FUNCTION_BLOCK FB_DXL_XL
VAR_INPUT 
	id : INT;
END_VAR
VAR  
	//communication en cours
	com_ongoing	: BOOL;
END_VAR
VAR CONSTANT
	//type du moteur
	XL430:USINT:=2;
	AX12A:USINT:=1;
	
	motor_type : USINT:=XL430;
END_VAR

//author: Alec Horth
//mail  : horth.alec@gmail.com

METHOD PRIVATE _end_communication : BOOL
VAR_IN_OUT
	run:BOOL; // arrête la variable qui maintient la fonction en vie 
	started:BOOL; // arrête la variable qui indique que la fonction possède un token
END_VAR
VAR_INST
	pulse : F_TRIG;
	once : bool;
END_VAR
// front descendant activé par le script python et désactivé par la fonction _send()
// confirme que la commande à bien été envoyée
pulse(CLK:=G_DXL.bDone AND started, Q=>);

IF pulse.Q THEN 
	//permet de lancer cette fonction une seule fois, sinon elle relance un cycle de façon involontaire 
	once := TRUE;
END_IF

IF once THEN
	// libère le token
	G_DXL.bToken := G_DXL.iOPEN_TOKEN;
	com_ongoing := FALSE;
	run := FALSE;
	_end_communication := TRUE;
	started := FALSE;
	once := FALSE;
ELSE
	_end_communication := FALSE;
END_IF
END_METHOD

METHOD PRIVATE _send : BOOL
VAR_INPUT
END_VAR
VAR_INST
	once :BOOL; // assure que la commande n'est envoyé qu'une fois
END_VAR
IF G_DXL.bDone THEN 	//confirmation d'acquisition de la commande du script python
	G_DXL.bRun := FALSE; //indique au script python que le message est passé
ELSIF NOT G_DXL.bDone AND NOT once THEN // si la commande n'a pas encore été envoyé, lance la commande
	once := TRUE;
	G_DXL.bRun := TRUE;
END_IF

IF NOT com_ongoing THEN // permet de relancer des commandes lorsque le token est rendu
	once := FALSE;
END_IF
END_METHOD

METHOD PRIVATE _start_communication : BOOL
VAR_IN_OUT
	started:BOOL; //maintient la fonction active tant que le token n'est pas rendu
END_VAR
IF ((G_DXL.bToken = G_DXL.iOPEN_TOKEN OR G_DXL.bToken = id) AND NOT com_ongoing AND NOT G_DXL.bDone) OR started THEN // vérifie que tous les token soient libres
	// attribution du token
	started := TRUE; 
	G_DXL.bToken := id;
	// configure les commandes à envoyer avec le bon ID et le bon type du moteur
	G_DXL.iID := id;
	G_DXL.usiMotor_type := motor_type;
	com_ongoing := TRUE; 
	_start_communication := TRUE;	
ELSE 
	_start_communication := FALSE;
END_IF
END_METHOD

METHOD private BASE_EXEMPLE_FUTUR_MODIF_SEND : BOOL
VAR_INPUT
	EN			:BOOL; // un front montant change le taux d'accélération du moteur
	
	//--------------TO DO---------------
	parametre1	:usint;
	parametre2	:INT;
	//----------------------------------

END_VAR
VAR_OUTPUT
	done		:BOOL; //la commande est envoyée, passe à False si EN passe aussi à False
END_VAR
VAR_INST 
	bRun 		:BOOL;
	rtrigPulse 	:R_TRIG;
	bDone_pulse :BOOL;
	bStarted 	:BOOL;
END_VAR
// IL EST POSSIBLE DE MODIFIER LES SECTION "TO DO", LE RESTE NE DOIT PAS ÊTRE MODIFIE

//Activation de la fonction
rtrigPulse(CLK:=EN, Q=>);

IF rtrigPulse.Q THEN
	//Si une autre fonction est déjà en cours de traitement (token déjà pris) cette fonction ne peut pas être effectuée
	//La variable run garde l'ordre d'activation en mémoire et lance la fonction dès que le token est libéré
	bRun := TRUE;
END_IF

IF bRun THEN
	IF _start_communication(started:=bStarted) THEN 	//vérifie si les tokens sont libérés 
		
		//--------------TO DO---------------
		G_DXL.usiFonction := G_DXL.usiGOAL_ACCELERATION; 	// choix de la commande à envoyer		
		G_DXL.usiAcceleration 	:= parametre1;				//paramètre 1
		G_DXL.iSpeed    		:= parametre2;				//paramètre 2 
		//----------------------------------
		
		
		bDone_pulse := _end_communication(run:=bRun, started:=bStarted) AND EN;	//libère le token une fois que la commande est lancée
		_send();																//Envoi de la commande au moteur
	END_IF
END_IF;

IF bDone_pulse AND EN THEN														//Affiche le status d'excution de la fonction
	done := EN;																	//tant que EN est à True
ELSIF bDone_pulse AND NOT EN THEN
	bDone_pulse := FALSE;
END_IF
END_METHOD

METHOD get_load 
VAR_INPUT
	EN:BOOL; 	// ouvre un canal de transmission avec le moteur 
END_VAR
VAR_OUTPUT
	load:INT; 	// le moteur renvoie le torque qu'il emet à travers le canal (voir dans la méthode pour + d'infos)
				//(AX12A) 0-1023 torque est dans le sens inverse des aiguilles d'une montre, entre 1024 et 2047 le torque est dans le sens des aiguilles d'une montre
				//(XL430) +- 1000 pour mille du torque maximum si la valeur est positive => le torque est dans le sens inverse des aiguilles d'une montre
	done:bool;
END_VAR
VAR_inst 
	run :BOOL;
	pulse : R_TRIG;
	started: BOOL;
END_VAR
//ouvre le canal de transmission
pulse(CLK:=EN, Q=>);

IF pulse.Q THEN
	//Si une autre fonction est déjà en cours de traitement (token déjà pris) le canal ne peut pas être ouvert
	//La variable run garde l'ordre d'activation en mémoire et ouvre le canal dès que le token est libéré
	run := TRUE;
END_IF

IF run THEN 
	IF _start_communication(started := started) THEN 	// Vérifie si le token est libre
		G_DXL.usiFonction := G_DXL.usiGET_PRESENT_LOAD;	// configure le canal à ouvrir
		G_DXL.bRun := TRUE;								// envoie la commande au script python
		load := G_DXL.iDxl_load;						// si le canal est ouvert, renvoie la valeur actuelle du torque émit pas le moteur
	END_IF
	IF NOT EN THEN
		G_DXL.bRun 	:= FALSE;						    //ferme le canal
		G_DXL.iDxl_load := -9000;						//remet une valeur par défault
		_end_communication(run:=run,started := started);//libère le token
	END_IF;
ELSE
	load := -9000;										//valeur par défaut
END_IF
END_METHOD

METHOD get_movement 
VAR_INPUT
	EN:BOOL; 	// ouvre un canal de transmission avec le moteur 
END_VAR
VAR_OUTPUT
	mouvement:BOOL; // le moteur renvoie si il est en mouvement(TRUE) ou non (FALSE)
END_VAR
VAR_INST 
	run :BOOL;
	pulse : R_TRIG;
	started: BOOL;
END_VAR
//ouvre le canal de transmission
pulse(CLK:=EN, Q=>);

IF pulse.Q THEN
	//Si une autre fonction est déjà en cours de traitement (token déjà pris) le canal ne peut pas être ouvert
	//La variable run garde l'ordre d'activation en mémoire et ouvre le canal dès que le token est libéré
	run := TRUE;
END_IF

IF run THEN 
	IF _start_communication(started := started) THEN 	// Vérifie si le token est libre
		G_DXL.usiFonction := G_DXL.usiGET_PRESENT_MOVEMENT;	// configure le canal à ouvrir
		G_DXL.bRun := TRUE;								// envoie la commande au script python
		mouvement := G_DXL.bDxl_movement;				// status du mouvement du moteur Dynamixel
	END_IF
	IF NOT EN THEN
		G_DXL.bRun 	:= FALSE;						    //ferme le canal
		G_DXL.bDxl_movement := 1;						//remet une valeur par défault
		_end_communication(run:=run,started := started);//libère le token
	END_IF;
ELSE
	mouvement := 1;										//valeur par défaut
END_IF
END_METHOD

METHOD get_position
VAR_INPUT
	EN:BOOL; 	// ouvre un canal de transmission avec le moteur 
END_VAR
VAR_OUTPUT
	position:DINT; //(AX12A sur 300 degrés)0-1023 ou (XL430 sur 360 degrés)0-4095 ou (XL430 en multitours)+- 1'048'575
END_VAR
VAR_INST 
	run :BOOL;
	pulse : R_TRIG;
	started: BOOL;
END_VAR
//ouvre le canal de transmission
pulse(CLK:=EN, Q=>);

IF pulse.Q THEN
	//Si une autre fonction est déjà en cours de traitement (token déjà pris) le canal ne peut pas être ouvert
	//La variable run garde l'ordre d'activation en mémoire et ouvre le canal dès que le token est libéré
	run := TRUE;
END_IF

IF run THEN 
	IF _start_communication(started := started) THEN 	// Vérifie si le token est libre
		G_DXL.usiFonction := G_DXL.usiGET_PRESENT_POSITION;	// configure le canal à ouvrir
		G_DXL.bRun := TRUE;								// envoie la commande au script python
		position := G_DXL.diDxl_position;				//(AX12A sur 300 degrés)0-1023 ou (XL430 sur 360 degrés)0-4095 ou (XL430 en multitours)+- 1'048'575
	END_IF
	IF NOT EN THEN
		G_DXL.bRun 	:= FALSE;						    //ferme le canal
		G_DXL.diDxl_position := -9000;					//remet une valeur par défault
		_end_communication(run:=run,started := started);//libère le token
	END_IF;
ELSE
	position := -9000;									//valeur par défaut
END_IF
END_METHOD

METHOD send_acceleration 
VAR_INPUT
	EN			:BOOL; // un front montant change le taux d'accélération du moteur
	acceleration:USINT;// acceleration de 0-100 (100 => acceleration instantanée)
	speed		:INT:=32767; // vitesse de pointe 0-32767
END_VAR
VAR_OUTPUT
	done		:BOOL; //la commande est envoyée, passe à False si EN passe aussi à False
END_VAR
VAR_INST 
	bRun 		:BOOL;
	rtrigPulse 	:R_TRIG;
	bDone_pulse :BOOL;
	bStarted 	:BOOL;
END_VAR
//Activation de la fonction
rtrigPulse(CLK:=EN, Q=>);

IF rtrigPulse.Q THEN
	//Si une autre fonction est déjà en cours de traitement (token déjà pris) cette fonction ne peut pas être effectuée
	//La variable run garde l'ordre d'activation en mémoire et lance la fonction dès que le token est libéré
	bRun := TRUE;
END_IF

IF bRun THEN
	IF _start_communication(started:=bStarted) THEN 								//vérifie si les tokens sont libérés 
		G_DXL.usiFonction := G_DXL.usiGOAL_ACCELERATION;								//Ecriture de la commande
		G_DXL.usiAcceleration := acceleration;
		G_DXL.iSpeed    := speed;
		bDone_pulse := _end_communication(run:=bRun, started:=bStarted) AND EN;	//libère le token une fois que la commande est lancée
		_send();																//Envoi de la commande au moteur
	END_IF
END_IF;

IF bDone_pulse AND EN THEN														//Affiche le status d'excution de la fonction
	done := EN;																	//tant que EN est à True
ELSIF bDone_pulse AND NOT EN THEN
	bDone_pulse := FALSE;
END_IF
END_METHOD

METHOD send_disable_torque
VAR_INPUT
	EN			:BOOL; // un front montant désactive le torque du moteur 
END_VAR
VAR_OUTPUT
	done		:BOOL; //la commande est envoyée, passe à False si EN passe aussi à False
END_VAR
VAR_INST 
	run 		:BOOL;
	pulse 		:R_TRIG;
	done_pulse 	:BOOL;
	started 	:BOOL;
END_VAR
//Activation de la fonction
pulse(CLK:=EN, Q=>);

IF pulse.Q THEN
	//Si une autre fonction est déjà en cours de traitement (token déjà pris) cette fonction ne peut pas être effectuée
	//La variable run garde l'ordre d'activation en mémoire et lance la fonction dès que le token est libéré
	run := TRUE;
END_IF

IF run THEN
	IF _start_communication(started:=started) THEN 								//vérifie si les tokens sont libérés 
		G_DXL.usiFonction := G_DXL.usiDISABLE_TORQUE;									//Ecriture de la commande
		done_pulse := _end_communication(run:=run, started:=started) AND EN;	//libère le token une fois que la commande est lancée
		_send();																//Envoi de la commande au moteur
	END_IF
END_IF;

IF done_pulse AND EN THEN														//Affiche le status d'excution de la fonction
	done := EN;																	//tant que EN est à True
ELSIF done_pulse AND NOT EN THEN
	done_pulse := FALSE;
END_IF
END_METHOD

METHOD send_enable_torque 
VAR_INPUT
	EN			:BOOL; // un front montant active le torque du moteur 
END_VAR
VAR_OUTPUT
	done		:BOOL; //la commande est envoyée, passe à False si EN passe aussi à False
END_VAR
VAR_INST 
	run 		:BOOL;
	pulse 		:R_TRIG;
	done_pulse 	:BOOL;
	started 	:BOOL;
END_VAR
//Activation de la fonction
pulse(CLK:=EN, Q=>);

IF pulse.Q THEN
	//Si une autre fonction est déjà en cours de traitement (token déjà pris) cette fonction ne peut pas être effectuée
	//La variable run garde l'ordre d'activation en mémoire et lance la fonction dès que le token est libéré
	run := TRUE;
END_IF

IF run THEN
	IF _start_communication(started:=started) THEN 								//vérifie si les tokens sont libérés 
		G_DXL.usiFonction := G_DXL.usiENABLE_TORQUE;									//Ecriture de la commande
		done_pulse := _end_communication(run:=run, started:=started) AND EN;	//libère le token une fois que la commande est lancée
		_send();																//Envoi de la commande au moteur
	END_IF
END_IF;

IF done_pulse AND EN THEN														//Affiche le status d'excution de la fonction
	done := EN;																	//tant que EN est à True
ELSIF done_pulse AND NOT EN THEN
	done_pulse := FALSE;
END_IF
END_METHOD

METHOD send_led_off 
VAR_INPUT
	EN			:BOOL; // un front montant éteint la led
END_VAR
VAR_OUTPUT
	done		:BOOL; //la commande est envoyée, passe à False si EN passe aussi à False
END_VAR
VAR_INST 
	run 		:BOOL;
	pulse 		:R_TRIG;
	done_pulse 	:BOOL;
	started 	:BOOL;
END_VAR
//Activation de la fonction
pulse(CLK:=EN, Q=>);

IF pulse.Q THEN
	//Si une autre fonction est déjà en cours de traitement (token déjà pris) cette fonction ne peut pas être effectuée
	//La variable run garde l'ordre d'activation en mémoire et lance la fonction dès que le token est libéré
	run := TRUE;
END_IF

IF run THEN
	IF _start_communication(started:=started) THEN 								//vérifie si les tokens sont libérés 
		G_DXL.usiFonction := G_DXL.usiLED_OFF;										//Ecriture de la commande
		done_pulse := _end_communication(run:=run, started:=started) AND EN;	//libère le token une fois que la commande est lancée
		_send();																//Envoi de la commande au moteur
	END_IF
END_IF;

IF done_pulse AND EN THEN														//Affiche le status d'excution de la fonction
	done := EN;																	//tant que EN est à True
ELSIF done_pulse AND NOT EN THEN
	done_pulse := FALSE;
END_IF
END_METHOD

METHOD send_led_on 
VAR_INPUT
	EN			:BOOL; // un front montant allume la led
END_VAR
VAR_OUTPUT
	done		:BOOL; //la commande est envoyée, passe à False si EN passe aussi à False
END_VAR
VAR_INST 
	run 		:BOOL;
	pulse 		:R_TRIG;
	done_pulse 	:BOOL;
	started 	:BOOL;
END_VAR
//Activation de la fonction
pulse(CLK:=EN, Q=>);

IF pulse.Q THEN
	//Si une autre fonction est déjà en cours de traitement (token déjà pris) cette fonction ne peut pas être effectuée
	//La variable run garde l'ordre d'activation en mémoire et lance la fonction dès que le token est libéré
	run := TRUE;
END_IF

IF run THEN
	IF _start_communication(started:=started) THEN 								//vérifie si les tokens sont libérés 
		G_DXL.usiFonction := G_DXL.usiLED_ON;											//Ecriture de la commande
		done_pulse := _end_communication(run:=run, started:=started) AND EN;	//libère le token une fois que la commande est lancée
		_send();																//Envoi de la commande au moteur
	END_IF
END_IF;

IF done_pulse AND EN THEN														//Affiche le status d'excution de la fonction
	done := EN;																	//tant que EN est à True
ELSIF done_pulse AND NOT EN THEN
	done_pulse := FALSE;
END_IF
END_METHOD

METHOD send_operating_mode 
VAR_INPUT
	EN			:BOOL; // active la fonction
	mode		:STRING; //‘position’ ou ‘position_angleMin_angleMax’ ou ‘extended position’ ou‘velocity' ou ‘PWM’ 
END_VAR
VAR_OUTPUT
	done		:BOOL; //la commande est envoyée, passe à False si EN passe aussi à False
END_VAR
VAR_INST 
	run 		:BOOL;
	pulse 		:R_TRIG;
	done_pulse 	:BOOL;
	started 	:BOOL;
END_VAR
//Activation de la fonction
pulse(CLK:=EN, Q=>);

IF pulse.Q THEN
	//Si une autre fonction est déjà en cours de traitement (token déjà pris) cette fonction ne peut pas être effectuée
	//La variable run garde l'ordre d'activation en mémoire et lance la fonction dès que le token est libéré
	run := TRUE;
END_IF

IF run THEN
	IF _start_communication(started:=started) THEN 								//vérifie si les tokens sont libérés 
		G_DXL.usiFonction := G_DXL.usiOPERATING_MODE;									//Ecriture de la commande
		G_DXL.sMode := mode;
		done_pulse := _end_communication(run:=run, started:=started) AND EN;	//libère le token une fois que la commande est lancée
		_send();																//Envoi de la commande au moteur
	END_IF
END_IF;

IF done_pulse AND EN THEN														//Affiche le status d'excution de la fonction
	done := EN;																	//tant que EN est à True
ELSIF done_pulse AND NOT EN THEN
	done_pulse := FALSE;
END_IF
END_METHOD

METHOD send_position 
VAR_INPUT
	EN			:BOOL; // un front montant donne une nouvelle position au moteur à atteindre 
	position	:DINT; //(AX12A sur 300 degrés)0-1023 ou (XL430 sur 360 degrés)0-4095 ou (XL430 en multitours)+- 1'048'575
	vitesse		:INT;  //(AX12A)0-1023 ou (XL430)0-1023 
END_VAR
VAR_OUTPUT
	done		:BOOL; //la commande est envoyée, passe à False si EN passe aussi à False
END_VAR
VAR_INST 
	run 		:BOOL;
	pulse 		:R_TRIG;
	done_pulse 	:BOOL;
	started 	:BOOL;
END_VAR
//Activation de la fonction
pulse(CLK:=EN, Q=>);

IF pulse.Q THEN
	//Si une autre fonction est déjà en cours de traitement (token déjà pris) cette fonction ne peut pas être effectuée
	//La variable run garde l'ordre d'activation en mémoire et lance la fonction dès que le token est libéré
	run := TRUE;
END_IF

IF run THEN
	IF _start_communication(started:=started) THEN 								//vérifie si les tokens sont libérés 
		G_DXL.usiFonction := G_DXL.usiGOAL_POSITION;									//Ecriture de la commande
		G_DXL.diPosition := position;
		G_DXL.iSpeed    := vitesse;
		done_pulse := _end_communication(run:=run, started:=started) AND EN;	//libère le token une fois que la commande est lancée
		_send();																//Envoi de la commande au moteur
	END_IF
END_IF;

IF done_pulse AND EN THEN														//Affiche le status d'excution de la fonction
	done := EN;																	//tant que EN est à True
ELSIF done_pulse AND NOT EN THEN
	done_pulse := FALSE;
END_IF
END_METHOD

METHOD send_reset_position 
VAR_INPUT
	EN			:BOOL; // un front montant réinitialise la position du moteur sur 360 degrés
END_VAR
VAR_OUTPUT
	done		:BOOL; //la commande est envoyée, passe à False si EN passe aussi à False
END_VAR
VAR_INST 
	run 		:BOOL;
	pulse 		:R_TRIG;
	done_pulse 	:BOOL;
	started 	:BOOL;
END_VAR
//Activation de la fonction
pulse(CLK:=EN, Q=>);

IF pulse.Q THEN
	//Si une autre fonction est déjà en cours de traitement (token déjà pris) cette fonction ne peut pas être effectuée
	//La variable run garde l'ordre d'activation en mémoire et lance la fonction dès que le token est libéré
	run := TRUE;
END_IF

IF run THEN
	IF _start_communication(started:=started) THEN 								//vérifie si les tokens sont libérés 
		G_DXL.usiFonction := G_DXL.usiRESET_POSITION;									//Ecriture de la commande
		done_pulse := _end_communication(run:=run, started:=started) AND EN;	//libère le token une fois que la commande est lancée
		_send();																//Envoi de la commande au moteur
	END_IF
END_IF;

IF done_pulse AND EN THEN														//Affiche le status d'excution de la fonction
	done := EN;																	//tant que EN est à True
ELSIF done_pulse AND NOT EN THEN
	done_pulse := FALSE;
END_IF
END_METHOD

METHOD send_stop_position 
VAR_INPUT
	EN			:BOOL; // un front montant arrête le moteur à sa position actuelle
	reset 		:BOOL; // reset la position 
END_VAR
VAR_OUTPUT
	done		:BOOL; //la commande est envoyée, passe à False si EN passe aussi à False
END_VAR
VAR_INST 
	run 		:BOOL;
	pulse 		:R_TRIG;
	done_pulse 	:BOOL;
	started 	:BOOL;
END_VAR
//Activation de la fonction
pulse(CLK:=EN, Q=>);

IF pulse.Q THEN
	//Si une autre fonction est déjà en cours de traitement (token déjà pris) cette fonction ne peut pas être effectuée
	//La variable run garde l'ordre d'activation en mémoire et lance la fonction dès que le token est libéré
	run := TRUE;
END_IF

IF run THEN
		IF _start_communication(started:=started) THEN 								//vérifie si les tokens sont libérés 
		G_DXL.usiFonction := G_DXL.usiSTOP_POSITION;										//Ecriture de la commande
		G_DXL.bReset	   := reset;
		done_pulse := _end_communication(run:=run, started:=started) AND EN;		//libère le token une fois que la commande est lancée
		_send();																	//Envoi de la commande au moteur
	END_IF
END_IF;

IF done_pulse AND EN THEN														//Affiche le status d'excution de la fonction
	done := EN;																	//tant que EN est à True
ELSIF done_pulse AND NOT EN THEN
	done_pulse := FALSE;
END_IF
END_METHOD

METHOD send_velocity 
VAR_INPUT
	EN			:BOOL; // un front montant donne une nouvelle vitesse au moteur en mode velocity
	vitesse		:INT;  //(XL430)+-1023 
END_VAR
VAR_OUTPUT
	done		:BOOL; //la commande est envoyée, passe à False si EN passe aussi à False
END_VAR
VAR_INST 
	run 		:BOOL;
	pulse 		:R_TRIG;
	done_pulse 	:BOOL;
	started 	:BOOL;
END_VAR
//Activation de la fonction
pulse(CLK:=EN, Q=>);

IF pulse.Q THEN
	//Si une autre fonction est déjà en cours de traitement (token déjà pris) cette fonction ne peut pas être effectuée
	//La variable run garde l'ordre d'activation en mémoire et lance la fonction dès que le token est libéré
	run := TRUE;
END_IF

IF run THEN
	IF _start_communication(started:=started) THEN 								//vérifie si les tokens sont libérés 
		G_DXL.usiFonction := G_DXL.usiGOAL_VELOCITY;									//Ecriture de la commande
		G_DXL.iSpeed    := vitesse;
		done_pulse := _end_communication(run:=run, started:=started) AND EN;	//libère le token une fois que la commande est lancée
		_send();																//Envoi de la commande au moteur
	END_IF
END_IF;

IF done_pulse AND EN THEN														//Affiche le status d'excution de la fonction
	done := EN;																	//tant que EN est à True
ELSIF done_pulse AND NOT EN THEN
	done_pulse := FALSE;
END_IF
END_METHOD

END_FUNCTION_BLOCK

(* stored: Version 1.1.0.1, ProductVersion 3.1.4024.12
   POU FB_DXL_XL: Id {2fdf5cc2-b098-424e-83c3-4e77bc6dfd2d}, SpecialFunc None
   Folder Envoi de commande (send): Id {825da9a6-1c3a-4f2f-9fb9-714b3641e950}
   Folder Fonctions internes: Id {819cbe36-25bb-4ef2-96c3-434f5e487d5c}
   Folder Reception d'informations (get): Id {e5ae8f8d-5230-4a2e-b2c2-1a01411e9520}
   Method _end_communication: Id {27177c34-6286-4140-bf5e-b8354e9049d4}
   Method _send: Id {38bdecc9-ecdd-4927-a973-c04f4673691e}
   Method _start_communication: Id {a7cf3886-121b-40c8-b3a6-e3d3f47f28fb}
   Method BASE_EXEMPLE_FUTUR_MODIF_SEND: Id {1c36c76b-a1e5-46cf-8278-7f3c5ab40023}
   Method get_load: Id {21150bce-726a-4f0c-b4c8-46ec650f5483}
   Method get_movement: Id {ab7af862-c94f-4b9e-89b2-995f754df3b6}
   Method get_position: Id {cf91e5cc-e978-4b65-8401-7d6a0b9b22d2}
   Method send_acceleration: Id {48fba966-1a24-4ff8-bfa9-92ca41798324}
   Method send_disable_torque: Id {27883b3b-620d-4452-ae1b-4d32ba2db699}
   Method send_enable_torque: Id {f6a15309-f08e-4149-9428-9cb9ebdf9ce6}
   Method send_led_off: Id {fbb44103-6f34-4682-841e-4170ccfac625}
   Method send_led_on: Id {93af1fae-070a-4dce-8f8b-8848afa127d9}
   Method send_operating_mode: Id {caa60429-e6a5-481b-b8b1-19d531a9f531}
   Method send_position: Id {ab93f21b-34e6-40af-8906-b7ea724d4789}
   Method send_reset_position: Id {6cf41c03-f680-4e4b-aac9-cf81cde2d7cd}
   Method send_stop_position: Id {39e13640-68dc-4d96-b523-24d9f7fc6ae9}
   Method send_velocity: Id {7090bb15-5b9f-4f0b-9001-d1a9131d985b} *)
